# EPICS StreamDevice protocol: home/outgas-ioc/modules/Pfeiffer-Controller-Device-Support/protocols/tpg_protocols.proto
Terminator = CR;

getModelNumber {
    out "AYT"; #<ARG> = Consists up to fifteen ASCII characters representing the current model number.
    in "\x06";
    out "\x05";
    in "%s";
}

getGaugePressure1 {
    out "PR1";
    in "\x06";
    out "\x05";
    in "%*[\n]0,%f";
}
